FUNCTION_BLOCK ILOCK_FB_RS_AX (* Realizes a bistable reset-dominat latch with AX interface and AX2 Interlock *)
  (* Standard: 61499-1; Description: Copyright (c) 2026 HR Agrartechnik GmbH This program and the accompanying materials are made available under the terms of the Eclipse Public License 2.0 which is available at https://www.eclipse.org/legal/epl-2.0/ SPDX-License-Identifier: EPL-2.0 *)
  (* Version 1.0, 2026-05-07, Gemini CLI, HR Agrartechnik GmbH, initial version *)
  PACKAGE logiBUS::signalprocessing::interlock;
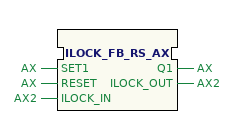
  SOCKETS
    SET1 : adapter::types::unidirectional::AX; (* Set *)
    RESET : adapter::types::unidirectional::AX; (* Reset *)
    ILOCK_IN : adapter::types::bidirectional::AX2; (* Interlock from above *)
  END_SOCKETS
  PLUGS
    Q1 : adapter::types::unidirectional::AX; (* Output *)
    ILOCK_OUT : adapter::types::bidirectional::AX2; (* Interlock to below *)
  END_PLUGS
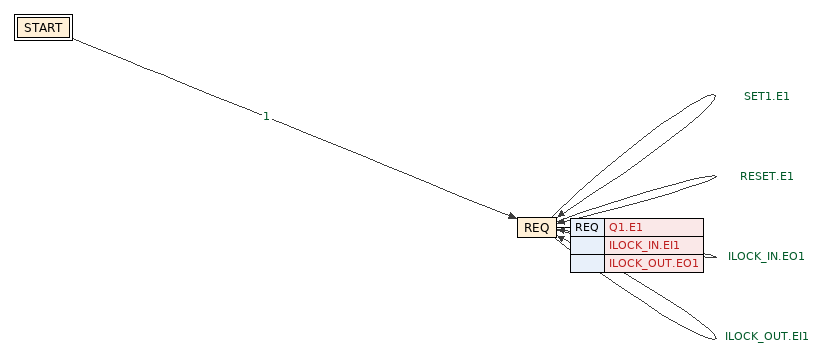
  EC_STATES
    START;
    REQ : REQ -> Q1.E1, -> ILOCK_IN.EI1, -> ILOCK_OUT.EO1;
  END_STATES
  EC_TRANSITIONS
    START TO REQ := 1;
    REQ TO REQ := SET1.E1;
    REQ TO REQ := RESET.E1;
    REQ TO REQ := ILOCK_IN.EO1;
    REQ TO REQ := ILOCK_OUT.EI1;
  END_TRANSITIONS
  ALGORITHM REQ IN ST:
	(* Reset-dominant logic: Q = (SET OR Q) AND NOT (RESET OR INTERLOCKS) *)
	Q1.D1 := (SET1.D1 OR Q1.D1) AND NOT (RESET.D1 OR ILOCK_IN.DO1 OR ILOCK_OUT.DI1);

	(* Propagate Reset signal to neighbors *)
	ILOCK_IN.DI1 := RESET.D1 OR ILOCK_OUT.DI1;
	ILOCK_OUT.DO1 := RESET.D1 OR ILOCK_IN.DO1;
  END_ALGORITHM
END_FUNCTION_BLOCK
